// TwinCAT 3 PLC project ads_com_sample
// ProgramVersion: 3.1.4024.0
// libraries:
//   Tc2_Standard, * (Beckhoff Automation GmbH)
//   Tc2_System, * (Beckhoff Automation GmbH)
//   Tc2_Utilities, * (Beckhoff Automation GmbH)
//   Tc3_Module, * (Beckhoff Automation GmbH)
// project tree:
//   DUTs/ ST_sample.TcDUT
//   / PlcTask.TcTTO
//   POUs/ ADS_Read.TcPOU, ADS_Write.TcPOU, EIP.TcPOU
// real-time tasks:
//   TASK PlcTask: cycle T#10ms, priority 20, ADS port 350
// I/O:
//   DEVICE Device 1 (EtherCAT), AmsNetId 5.143.107.166.2.1
//     Term 1 (EK1200) [EK1200-7000 EtherCAT Power supply (1,5A E-Bus)]
//       Term 2 (EL6652) [EL6652 EtherNet/IP Scanner (Master)]
//       Term 3 (EL9011) [EL9011 End Terminal]
//   DEVICE Device 2 (NOV-DP-RAM)
//   DEVICE Device 3 (CX7000), AmsNetId 5.143.107.166.4.1
//     Term 1 (CX7028) [CX7028-0000-0118]
//       modules: Module 1 (DIO_2x), Module 3 (DIO_2x), Module 5 (DI_2x), Module 7 (DI_2x)
//   DEVICE Device 4 (COM Port)
//   DEVICE Device 5 (COM Port)
//   DEVICE Device 6 (ECAT EIP Scanner (EL6652)), AmsNetId 5.143.107.166.7.1
//     Box 5 (Box 1 (TC EtherNet/IP Slave)) // <INFO> </INFO> <EDS> C:\TwinCAT\3.1\Config\Io\EtherNetIP\Box 1 (TC EtherNet_IP Slave)_20240808_104409.eds </EDS>
// variable links:
//   ads_com_sample/ads_com_sample Instance <-> Device 6 (ECAT EIP Scanner (EL6652))/Box 5 (Box 1 (TC EtherNet/IP Slave))
//     PlcTask Inputs/EIP.eip_input <-> Connection 1 (Input/Output)/Inputs/Assembly 1 / Outputs / values
//     PlcTask Inputs/EIP.eip_input @bit {8..504 step 8} <-> Connection 1 (Input/Output)/Inputs/Assembly 1 / Outputs / values_{1..63}  (63 links)
//     PlcTask Outputs/EIP.eip_output <-> Connection 1 (Input/Output)/Outputs/Assembly 1 / Inputs / values
//     PlcTask Outputs/EIP.eip_output @bit {8..504 step 8} <-> Connection 1 (Input/Output)/Outputs/Assembly 1 / Inputs / values_{1..63}  (63 links)

CONFIGURATION ads_com_sample
    RESOURCE PLC ON TwinCAT3
        TASK PlcTask(INTERVAL := T#10ms, PRIORITY := 20);
        PROGRAM ADS_Read WITH PlcTask : ADS_Read;
        PROGRAM ADS_Write WITH PlcTask : ADS_Write;
        PROGRAM EIP WITH PlcTask : EIP;
    END_RESOURCE
END_CONFIGURATION

// ---- DUTs/ST_sample.TcDUT
TYPE ST_sample :
STRUCT
	title : STRING;
	id : UINT;
	datetime : DT;
END_STRUCT
END_TYPE

// ---- POUs/ADS_Read.TcPOU
PROGRAM ADS_Read
VAR
    fbReadInd    : ADSREADINDEX := (MINIDXGRP := 16#8E000000);(* Indication function block instance *)
    fbReadRes    : ADSREADRES;(* Response function block instance *)
    sNetId       : T_AmsNetID;
    nPort        : T_AmsPort := 851;
    nInvokeId    : UDINT;
    nIdxGrp      : UDINT;
    nIdxOffs     : UDINT;
    cbLength     : UDINT;(* Requested read data/buffer byte size *)
    cbRead       : UDINT;(* Returned read data/buffer byte size *)
    pRead        : PVOID;(* Pointer to returned read data/buffer *)
    nErrID       : UDINT;(* Read indication result error code *)
    nCounter     : INT;(* Server data *)
	stSample 	 : ST_sample;
	fbSystemTime   : GETSYSTEMTIME;
    timeAsFileTime : T_FILETIME;
    timeAsDT       : DT;
	

END_VAR

fbReadRes( RESPOND := FALSE );(* Reset response function block *) 
 fbReadInd( CLEAR := FALSE );(* Trigger indication function block *) 
 IF fbReadInd.VALID THEN(* Check for new indication *) 
 
      sNetID := fbReadInd.NETID; 
      nPort := fbReadInd.PORT; 
      nInvokeID := fbReadInd.INVOKEID; 
      nIdxGrp := fbReadInd.IDXGRP; 
      nIdxOffs := fbReadInd.IDXOFFS; 
      cbLength := fbReadInd.LENGTH; 
 
      cbRead := 0; 
      pRead := 0; 
      nErrID     := DEVICE_SRVNOTSUPP; 
 
      
     CASE nIdxGrp OF 
          (*------------------------------------------------------------------------------------*) 
          16#8E000001: 
               CASE nIdxOffs OF 
                    0:(* Increment counter value *) 
                         IF cbLength >= SIZEOF(nCounter) THEN 
                              nCounter := nCounter + 1; 
                              cbRead := SIZEOF(nCounter); 
                              pRead := ADR(nCounter); 
                              nErrID := NOERR; 
                         ELSE (* ADS error (example): Invalid size *) 
                              nErrID := DEVICE_INVALIDSIZE; 
                         END_IF 
               ELSE (* ADS error (example): Invalid index offset *) 
                    nErrID := DEVICE_INVALIDOFFSET; 
               END_CASE 
          (*------------------------------------------------------------------------------------*) 
          16#8E000002: 
               CASE nIdxOffs OF 
                    0:(* Decrement counter value *) 
                         IF cbLength >= SIZEOF(nCounter) THEN 
                              nCounter := nCounter - 1; 
                              cbRead := SIZEOF(nCounter); 
                              pRead := ADR(nCounter); 
                              nErrID := NOERR; 
                         ELSE(* ADS error (example): Invalid size *) 
                              nErrID := DEVICE_INVALIDSIZE; 
                         END_IF 
               ELSE (* ADS error (example): Invalid index offset *) 
                    nErrID := DEVICE_INVALIDOFFSET; 
               END_CASE 
          (*------------------------------------------------------------------------------------*) 
          16#8E000003: 
               CASE nIdxOffs OF 
                    0:(* Reset counter value *) 
                         IF cbLength >= SIZEOF(nCounter) THEN 
                              nCounter := 0; 
                              cbRead := SIZEOF(nCounter); 
                              pRead := ADR(nCounter); 
                              nErrID := NOERR; 
                         ELSE(* ADS error (example): Invalid size *) 
                              nErrID := DEVICE_INVALIDSIZE; 
                         END_IF 
               ELSE (* ADS error (example): ervice is not supported by server *) 
                    nErrID := DEVICE_SRVNOTSUPP; 
               END_CASE 
			   
			16#8E000004:
				CASE nIdxOffs OF
					0:(* Modify structured variable *) 
                         IF cbLength >= SIZEOF(stSample) THEN 
                            stSample.id := stSample.id + 1;
							stSample.title := 'TEST';
							fbSystemTime( timeLoDW=>timeAsFileTime.dwLowDateTime, timeHiDW=>timeAsFileTime.dwHighDateTime );
							stSample.datetime := FILETIME_TO_DT( timeAsFileTime );
                              cbRead := SIZEOF(stSample); 
                              pRead := ADR(stSample); 
                              nErrID := NOERR; 
                         ELSE(* ADS error (example): Invalid size *) 
                              nErrID := DEVICE_INVALIDSIZE; 
                         END_IF 
				END_CASE
 
     ELSE (* ADS error (example): Invalid index group *) 
          nErrID := DEVICE_INVALIDGRP; 
     END_CASE 
      
     fbReadRes(     NETID := sNetID, 
                    PORT := nPort, 
                    INVOKEID := nInvokeID, 
                    LEN := cbRead, 
                    DATAADDR := pRead, 
                    RESULT := nErrID, 
                    RESPOND := TRUE );(* Send read response *) 
                     
     fbReadInd( CLEAR := TRUE ); (* Clear indication entry *) 
END_IF

END_PROGRAM

// ---- POUs/ADS_Write.TcPOU
PROGRAM ADS_Write
VAR
   fbWriteInd  : ADSWRITEINDEX;
   fbWriteRes  : ADSWRITERES;
   sNetId      : T_AmsNetID;
   nPort       : T_AmsPort;
   nInvokeId   : UDINT;
   nIdxGrp     : UDINT;
   nIdxOffs    : UDINT;
   cbWrite     : UDINT;(* Byte size of written data *)
   pWrite      : PVOID;(* Pointer to written data buffer *)
   nResult     : UDINT;(* Write indication result error code *)
   arrInt      : ARRAY[0..9] OF INT;(* Server data *)
END_VAR

fbWriteRes( RESPOND := FALSE );(* Reset response function block *)
fbWriteInd( CLEAR := FALSE );(* Trigger indication function block *)
IF ( fbWriteInd.VALID ) THEN
   
   sNetId       := fbWriteInd.NETID;
   nPort        := fbWriteInd.PORT;
   nInvokeId    := fbWriteInd.INVOKEID;
   nIdxGrp      := fbWriteInd.IDXGRP;
   nIdxOffs     := fbWriteInd.IDXOFFS;
   cbWrite      := fbWriteInd.LENGTH;
   pWrite       := fbWriteInd.DATAADDR;
   nResult      := DEVICE_SRVNOTSUPP;

   CASE nIdxGrp OF
      16#80000005:
         CASE nIdxOffs OF
            16#00000000:
               IF cbWrite <= SIZEOF( arrInt ) THEN
                  MEMCPY( ADR( arrInt ), pWrite, MIN( cbWrite, SIZEOF(arrInt) ) );
                  nResult := NOERR;
               ELSE(* ADS error (example): Invalid size *)
                  nResult := DEVICE_INVALIDSIZE;
               END_IF
         ELSE(* ADS error (example): Invalid index offset *)
            nResult := DEVICE_INVALIDOFFSET;
         END_CASE
   ELSE(* ADS error (example): Invalid index group *)
      nResult := DEVICE_INVALIDGRP;
   END_CASE

   fbWriteRes( NETID := sNetId,
            PORT := nPort,
            INVOKEID := nInvokeId,
            RESULT := nResult,
            RESPOND := TRUE ); (* Send write response *)

   fbWriteInd( CLEAR := TRUE ); (* Clear indication entry *)
END_IF

END_PROGRAM

// ---- POUs/EIP.TcPOU
PROGRAM EIP
VAR
	eip_input AT%I* 	: ARRAY[0..63] OF BYTE;
	eip_output AT%Q* 	: ARRAY[0..63] OF BYTE;
	
	i :UINT;
	counter : UINT;
	diff : BYTE;
END_VAR

IF counter > 255 THEN
	counter := 0;
ELSE
	counter := counter + 1;
END_IF

FOR i := 0 TO 63 DO
	eip_output[i] := UINT_TO_BYTE(counter);
END_FOR

diff := eip_output[1] - eip_input[1];

END_PROGRAM
